(* IEC 61131-3 sources: my-first-app/src, 8 files *)

(* ---- types.st ---- *)
TYPE
    my_Struct : STRUCT
    my_BOOL: BOOL;
    my_int: INT;
    END_STRUCT;

END_TYPE

(* ---- myfunction.st ---- *)
FUNCTION myfunction : INT
    VAR_INPUT
    myIN: INT;
    END_VAR

    VAR_TEMP
    END_VAR
    ;

END_FUNCTION

FUNCTION myfunction_2 : INT
    VAR_INPUT
    myIN_2: INT;
    END_VAR

    ;

END_FUNCTION

(* ---- fb.st ---- *)
FUNCTION_BLOCK fb
    VAR_INPUT
        my_Input : LREAL;
    END_VAR
    VAR
        storage: LREAL;
    END_VAR

    ;
    END_FUNCTION_BLOCK

(* ---- myclass.st ---- *)
//NAMESPACE esempio

CLASS myclass
    VAR //default protected which means that they can be access from
        myStaticInt : INT;
    END_VAR

    VAR PUBLIC
        mypublic : INT;
    END_VAR

    VAR INTERNAL // can be access into the same namespace. If I do not have namespace, it is public.
        myInternal: INT;
    END_VAR

METHOD PUBLIC GetStaticInfo : INT
    GetStaticInfo:=myStaticInt;
END_METHOD

END_CLASS

(* ---- configuration.st ---- *)
CONFIGURATION MyConfiguration
    TASK Main(Interval := T#1000ms, Priority := 1);
    TASK task_2(Interval := T#1000ms, Priority := 1);
    TASK task_3(Interval := T#1000ms, Priority := 1);
    PROGRAM P1 WITH Main: MyProgram;
    PROGRAM P2 WITH task_2: MyProgram_2;
    PROGRAM P3 WITH task_3: MyProgram_3;

    VAR_GLOBAL

    END_VAR
END_CONFIGURATION

FUNCTION myfunction_3 : INT
    VAR_INPUT
    myIN_3: INT;
    ciao: INT;
    END_VAR

    ;

END_FUNCTION

(* ---- program.st ---- *)
PROGRAM MyProgram
    VAR_EXTERNAL

    END_VAR

    VAR
        myclassinstance: myclass;
    END_VAR

    VAR_TEMP

    END_VAR

    myclassinstance.mypublic := 1;
    myclassinstance.GetStaticInfo();
    myclassinstance.myInternal := 1;

    ;
END_PROGRAM

(* ---- program2.st ---- *)
PROGRAM MyProgram_2
    VAR_EXTERNAL

    END_VAR

    VAR

    END_VAR

    VAR_TEMP

    END_VAR

    // code here
    ;
END_PROGRAM

(* ---- program3.st ---- *)
PROGRAM MyProgram_3
    VAR_EXTERNAL

    END_VAR

    VAR

    END_VAR

    VAR_TEMP

    END_VAR

    // code here
    ;
END_PROGRAM
